// LS Electric XG5000 project: 71회예상2_3
// PLC NewPLC
// module base 0 slot 0: 입출력 모듈:XBC-DR20S (DC 24V 입력 12점, 릴레이 출력 8점)

PROGRAM NewProgram (task: 스캔 프로그램)

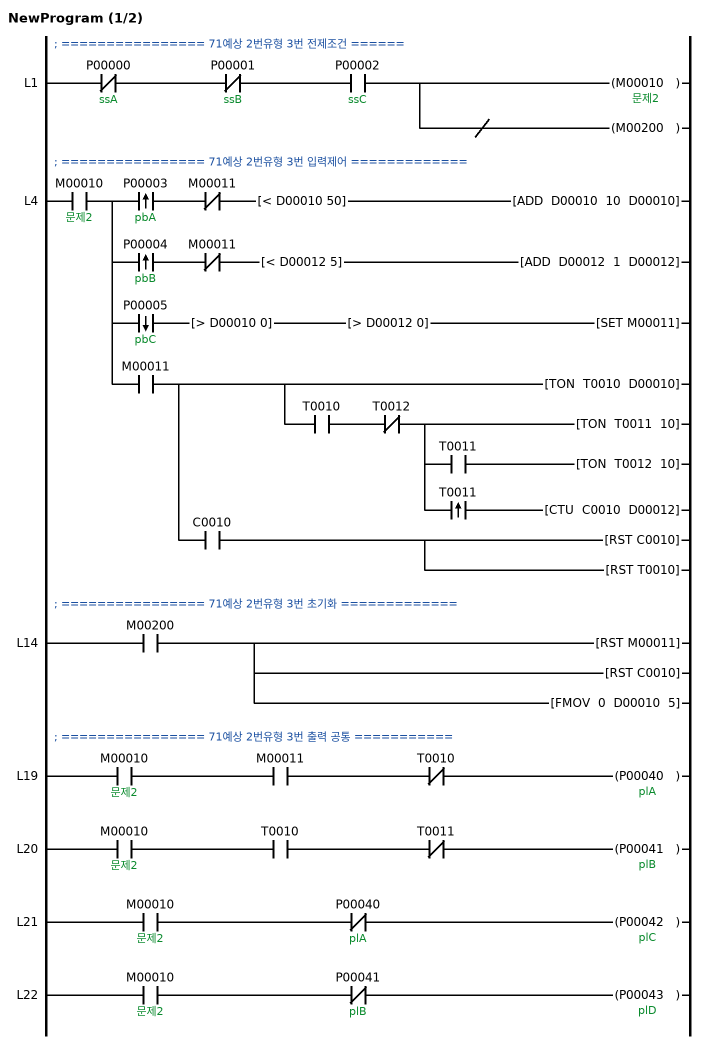
// ================ 71예상 2번유형 3번 전제조건 ======
; L1
LOAD NOT  P00000	// ssA
AND NOT   P00001	// ssB
AND       P00002	// ssC
OUT       M00010	// 문제2
NOT
OUT       M00200
// ================ 71예상 2번유형 3번 입력제어 =============
; L4
LOAD      M00010	// 문제2
MPUSH
ANDP      P00003	// pbA
AND NOT   M00011
AND<      D00010 50
ADD       D00010 10 D00010
MLOAD
ANDP      P00004	// pbB
AND NOT   M00011
AND<      D00012 5
ADD       D00012 1 D00012
MLOAD
ANDN      P00005	// pbC
AND>      D00010 0
AND>      D00012 0
SET       M00011
MPOP
AND       M00011
TON       T0010 D00010
MPUSH
AND       T0010
AND NOT   T0012
TON       T0011 10
MPUSH
AND       T0011
TON       T0012 10
MPOP
ANDP      T0011
CTU       C0010 D00012
MPOP
AND       C0010
RST       C0010
RST       T0010
// ================ 71예상 2번유형 3번 초기화 =============
; L14
LOAD      M00200
RST       M00011
RST       C0010
FMOV      0 D00010 5
// ================ 71예상 2번유형 3번 출력 공통 ===========
; L19
LOAD      M00010	// 문제2
AND       M00011
AND NOT   T0010
OUT       P00040	// plA
; L20
LOAD      M00010	// 문제2
AND       T0010
AND NOT   T0011
OUT       P00041	// plB
; L21
LOAD      M00010	// 문제2
AND NOT   P00040	// plA
OUT       P00042	// plC
; L22
LOAD      M00010	// 문제2
AND NOT   P00041	// plB
OUT       P00043	// plD

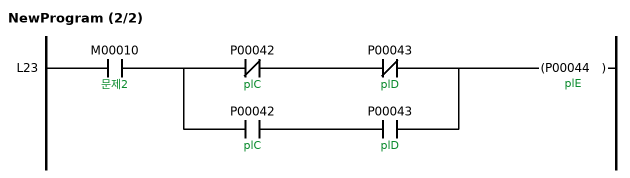
; L23
LOAD      M00010	// 문제2
LOAD NOT  P00042	// plC
AND NOT   P00043	// plD
LOAD      P00042	// plC
AND       P00043	// plD
OR LOAD
AND LOAD
OUT       P00044	// plE